
DATA_BLOCK db_Temp
//Присвоение переменных
STRUCT
    Old_P   :ARRAY [0..23] OF udt_Pipe;
END_STRUCT

BEGIN

END_DATA_BLOCK
